FUNCTION_BLOCK Real2Int (* Basic Function Block Type *)
  (* Standard: 61499-2 *)
  (* Version 0.0, 7/13/2023, Cheyan, Schneider Electric, Template *)
  PACKAGE Main;
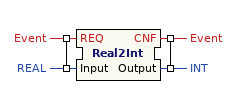
  EVENT_INPUT
    REQ WITH Input; (* Normal Execution Request *)
  END_EVENT
  EVENT_OUTPUT
    CNF WITH Output; (* Execution Confirmation *)
  END_EVENT
  VAR_INPUT
    Input : REAL; (* Input event qualifier *)
  END_VAR
  VAR_OUTPUT
    Output : INT; (* Output event qualifier *)
  END_VAR
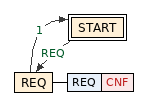
  EC_STATES
    START; (* Initial State *)
    REQ : REQ -> CNF; (* Normal execution *)
  END_STATES
  EC_TRANSITIONS
    START TO REQ := REQ;
    REQ TO START := 1;
  END_TRANSITIONS
  ALGORITHM REQ IN ST: (* Normally executed algorithm *)
;

IF Input = 0.0 THEN
	Output:=0;
ELSIF Input = 1.0 THEN
	Output:=1;
ELSIF Input = 2.0 THEN
	Output:=2;
ELSIF Input = 3.0 THEN
	Output:=3;
ELSIF Input = 4.0 THEN
	Output:=4;
ELSIF Input = 5.0 THEN
	Output:=5;
END_IF;
  END_ALGORITHM
END_FUNCTION_BLOCK
